INTERFACE I_AxisMoveRelative EXTENDS I_Base

METHOD MoveRelative : BOOL
VAR_INPUT
	Distance	  : LREAL;
	AbortPrevious : BOOL := TRUE;
END_VAR
END_METHOD

END_INTERFACE

(* stored: Version 1.1.0.1, ProductVersion 3.1.4026.18
   Itf I_AxisMoveRelative: Id {f7b139cd-e112-494e-acc8-6435afdcacf5}
   Method MoveRelative: Id {b528c3a7-3a1c-443e-bb1b-694bf2d690ed} *)
